TYPE ST_Filter :
STRUCT
    nHolderNumber : INT;
    nFilterNumber : INT;
    eFilterType : E_FilterType;
    eFilterMaterial : E_FilterMaterial;
    uFilterThickness : U_FilterThickness;
END_STRUCT
END_TYPE

(* stored: Version 1.1.0.1
   DUT ST_Filter: Id {60dc1f96-f95d-46a1-9aa8-1dcc67cd5427} *)
